(* IEC 61131-3 sources: eCockpitGit/test_project/src/%F%00 Library/%F%JSON/%POU%FB_JSONReader/%F%Structure, 12 files *)

(* ---- %METH%compareKeyName.st ---- *)
//Returns true if the inputted string is the same as the read string
METHOD compareKeyName : EStructType
VAR_INPUT
	name				:POINTER TO EASCII;
END_VAR
VAR
	posBuffer			:POINTER TO EASCII := lastKeyStart + 1;		//Buffer for key position
END_VAR
(*%!%__DELIMITER__%!%*)
IF ready AND_THEN selectedType = EStructType.object THEN
	WHILE posBuffer <= bufferADRMax DO
		CASE posBuffer^ OF
			EASCII.Null:
				IF name^ = EASCII.Null THEN
					compareKeyName		:=		lastValueType;
				END_IF
				EXIT;
			EASCII.DoubleQoute:
				IF checkNoBackSlash(checkPos:=posBuffer) THEN
					IF name^ = EASCII.Null THEN
						compareKeyName		:=		lastValueType;
					END_IF
					EXIT;
				END_IF
		END_CASE
		IF name^ <> posBuffer^ THEN
			IF posBuffer^ = EASCII.BackSlash THEN
				posBuffer				:=		posBuffer + 1;
				IF name^ <> posBuffer^ THEN
					EXIT;
				END_IF
			ELSE
				EXIT;
			END_IF
		END_IF
		name								:=		name + 1;
		posBuffer						:=		posBuffer + 1;
	END_WHILE
END_IF

(* ---- %METH%enterObjectArray.st ---- *)
//This method enters the last found object and sets it as the current object for searching
//Returns false, if not successfull
// |**Version**|**Author**| **Date** |**Changes**
// | 1         | NSN      | 04-06-18 | Creation
METHOD enterObjectArray :BOOL

(*%!%__DELIMITER__%!%*)
IF ready AND treeLevel < levelsMax THEN
	CASE lastValueType OF
		EStructType.object,EStructType.tArray:
			treeLevel			:=		treeLevel + 1;
			treeSelectedTypes[treeLevel]	:=		lastValueType;
			treeSelected[treeLevel]			:=		lastValueStart;
			treeSelectedArrayProg[treeLevel]:=		0;
			lastValueStart		:=		0;
			lastValueType		:=		EStructType.none;
			lastKeyStart		:=		0;
			enterObjectArray	:=		TRUE;
	END_CASE
END_IF

(* ---- %METH%exitObjectArray.st ---- *)
//This method exits the current object or array
//Returns none, when there are no more keys
// |**Version**|**Author**| **Date** |**Changes**
// | 1         | NSN      | 04-06-18 | Creation
METHOD exitObjectArray : BOOL
VAR
	inString		:BOOL;
	posBuffer		:POINTER TO EASCII := treeSelected[treeLevel] - 1;
	level			:WORD := 1;		//This value makes sure it doesn't return a key from inside another object
	keyFound		:BOOL;
END_VAR
(*%!%__DELIMITER__%!%*)
IF ready AND treeLevel > 1 THEN
	WHILE posBuffer >= bufferADROrg DO
		CASE posBuffer^ OF
			EASCII.DoubleQoute:
				IF checkNoBackSlash(checkPos:=posBuffer) THEN
					inString					:=		NOT(inString);
					IF keyFound AND NOT(inString) THEN
						lastKeyStart			:=		posBuffer;
					END_IF
				END_IF
			EASCII.Colon:
				IF NOT(inString) THEN
					keyFound					:=		TRUE;
				END_IF
			EASCII.CloseBraces,EASCII.SqBracketC:
				IF NOT(inString) THEN
					level						:=		level + 1;
				END_IF
			EASCII.OpenBraces,EASCII.SqBracketO,EASCII.Comma:
				IF NOT(inString) THEN
					IF level = 1 THEN
						lastValueStart			:=		treeSelected[treeLevel];
						lastValueType			:=		treeSelectedTypes[treeLevel];
						treeLevel				:=		treeLevel - 1;
						exitObjectArray			:=		TRUE;
						RETURN;
					ELSE
						level					:=		level - 1;
					END_IF
				END_IF
		END_CASE
		posBuffer								:=		posBuffer - 1;
	END_WHILE
END_IF

(* ---- %METH%exportSelection.st ---- *)
//This method outputs the start address and size of the currently selected object
//True when ok
// |**Version**|**Author**| **Date** |**Changes**
// | 1         | NSN      | 04-06-18 | Creation
METHOD exportSelection : BOOL
VAR_OUTPUT
	position		:POINTER TO EASCII;
	size			:DWORD;
END_VAR
VAR
	inString		:BOOL;
	posBuffer		:POINTER TO EASCII := treeSelected[treeLevel];
	level			:WORD;		//This value makes sure it doesn't return a key from inside another object
END_VAR
(*%!%__DELIMITER__%!%*)
IF ready AND treeLevel > 0 THEN
	position			:=		treeSelected[treeLevel];
	WHILE posBuffer < bufferADRMax DO
		CASE posBuffer^ OF
			EASCII.Null:EXIT;
			EASCII.DoubleQoute: IF checkNoBackSlash(checkPos:=posBuffer) THEN inString := NOT(inString); END_IF
			EASCII.CloseBraces,EASCII.SqBracketC: IF NOT(inString) THEN IF level > 1 THEN level := level - 1;ELSE EXIT; END_IF END_IF
			EASCII.OpenBraces,EASCII.SqBracketO: IF NOT(inString) THEN level := level + 1; END_IF
		END_CASE
		posBuffer												:=		posBuffer + 1;
	END_WHILE
	size				:=		posBuffer - position + 1;
	exportSelection		:=		TRUE;
END_IF

(* ---- %METH%findKey.st ---- *)
//This method finds the key of the given name in the object
//Returns cursor to where it was before if no tag is found
// |**Version**|**Author**| **Date** |**Changes**
// | 1         | NSN      | 04-06-18 | Creation
METHOD findKey : EStructType
VAR_INPUT
	name			:POINTER TO EASCII;		//Address of the name to find, only input string address or zero terminated byte array
END_VAR
VAR
	inString		:BOOL;
	nameBuffer		:POINTER TO EASCII;		//Buffer for cursor position
	posBuffer		:POINTER TO EASCII := treeSelected[treeLevel];
	level			:WORD;		//This value makes sure it doesn't return a key from inside another object
	foundKeyBuffer	:POINTER TO EASCII;
	slashDepth		:WORD;
END_VAR
(*%!%__DELIMITER__%!%*)
IF ready AND treeLevel > 0 AND treeSelectedTypes[treeLevel] = EStructType.object THEN
	WHILE posBuffer <= bufferADRMax DO
		CASE posBuffer^ OF
			EASCII.Null:EXIT;
			EASCII.DoubleQoute: IF checkNoBackSlash(checkPos:=posBuffer) THEN inString := NOT(inString); END_IF
			EASCII.CloseBraces,EASCII.SqBracketC: IF NOT(inString) THEN IF level > 1 THEN level := level - 1;ELSE EXIT; END_IF END_IF
			EASCII.SqBracketO: IF NOT(inString) THEN level := level + 1;END_IF
			EASCII.Comma,EASCII.OpenBraces:
				IF NOT(inString) THEN
					IF posBuffer^ = EASCII.OpenBraces THEN
						level									:=		level + 1;
					END_IF
					IF level = 1 THEN
						WHILE posBuffer <= bufferADRMax DO
							posBuffer							:=		posBuffer + 1;
							CASE posBuffer^ OF
								EASCII.Null:EXIT;
								EASCII.DoubleQoute:
									inString										:=		TRUE;
									nameBuffer										:=		name;
									foundKeyBuffer									:=		posBuffer;
									posBuffer										:=		posBuffer + 1;
									WHILE posBuffer <= bufferADRMax DO
										IF nameBuffer^ = EASCII.Null AND_THEN posBuffer^ = EASCII.DoubleQoute THEN
											WHILE posBuffer <= bufferADRMax DO
												CASE posBuffer^ OF
													EASCII.Null:EXIT;
													EASCII.DoubleQoute:
														IF checkNoBackSlash(checkPos:=posBuffer) THEN
															inString := NOT(inString);
														END_IF
													EASCII.Colon:
														IF NOT(inString) THEN
															findKey					:=		getType(valueFirstByte:=posBuffer + 1,valuePos=>lastValueStart);
															lastKeyStart			:=		foundKeyBuffer;
															lastValueType			:=		findKey;
															RETURN;
														END_IF
												END_CASE
												posBuffer							:=		posBuffer + 1;
											END_WHILE
										END_IF
										//Check for escape character
										IF nameBuffer^ = EASCII.DoubleQoute OR posBuffer^ = EASCII.BackSlash THEN
											posBuffer								:=		posBuffer + 1;
											IF posBuffer^ <> EASCII.DoubleQoute THEN
												posBuffer							:=		posBuffer - 1;
											END_IF
										END_IF
										IF posBuffer^ <> nameBuffer^ OR posBuffer^ = EASCII.Null THEN
											IF posBuffer^ = EASCII.DoubleQoute THEN
												IF checkNoBackSlash(checkPos:=posBuffer) THEN
													inString := NOT(inString);
												END_IF
											END_IF
											EXIT;
										END_IF
										nameBuffer									:=		nameBuffer + 1;
										posBuffer									:=		posBuffer + 1;
									END_WHILE
									EXIT;
							END_CASE
						END_WHILE
					END_IF
				END_IF
		END_CASE
		posBuffer																	:=		posBuffer + 1;
	END_WHILE
	findKey																			:=		EStructType.none;
END_IF

(* ---- %METH%nextArray.st ---- *)
//This method finds the next value in an array
//Returns none, when there are no more entries
// |**Version**|**Author**| **Date** |**Changes**
// | 1         | NSN      | 04-06-18 | Creation
METHOD nextArray : EStructType
VAR
	inString		:BOOL;
	posBuffer		:POINTER TO EASCII := lastValueStart;
	level			:WORD;		//This value makes sure it doesn't return a key from inside another object
END_VAR
(*%!%__DELIMITER__%!%*)
IF ready AND treeLevel > 0 AND treeSelectedTypes[treeLevel] = EStructType.tArray THEN
	IF lastValueStart = 0 THEN
		posBuffer									:=		treeSelected[treeLevel];
	ELSE
		level										:=		1;
	END_IF
	WHILE posBuffer <= bufferADRMax DO
		CASE posBuffer^ OF
			EASCII.Null:EXIT;
			EASCII.DoubleQoute: IF checkNoBackSlash(checkPos:=posBuffer) THEN inString := NOT(inString); END_IF
			EASCII.CloseBraces,EASCII.SqBracketC: IF NOT(inString) THEN IF level > 1 THEN level := level - 1;ELSE EXIT; END_IF END_IF
			EASCII.OpenBraces: IF NOT(inString) THEN level := level + 1;END_IF
			EASCII.Comma,EASCII.SqBracketO:
				IF NOT(inString) THEN
					IF posBuffer^ = EASCII.SqBracketO THEN
						level						:=		level + 1;
					END_IF
					IF level = 1 THEN
						nextArray					:=		getType(valueFirstByte:=posBuffer + 1,valuePos=>lastValueStart);
						lastValueType				:=		nextArray;
						treeSelectedArrayProg[treeLevel]	:=		treeSelectedArrayProg[treeLevel] + 1;
						RETURN;
					END_IF
				END_IF
		END_CASE
		posBuffer									:=		posBuffer + 1;
	END_WHILE
	nextArray										:=		EStructType.none;
END_IF

(* ---- %METH%nextKey.st ---- *)
//This method finds the next key/value pair in the current object
//Returns none, when there are no more keys
// |**Version**|**Author**| **Date** |**Changes**
// | 1         | NSN      | 04-06-18 | Creation
METHOD nextKey : EStructType
VAR
	inString		:BOOL;
	posBuffer		:POINTER TO EASCII := lastKeyStart;
	level			:WORD;		//This value makes sure it doesn't return a key from inside another object
	foundKeybuffer	:POINTER TO EASCII;
END_VAR
(*%!%__DELIMITER__%!%*)
IF ready AND treeLevel > 0 AND treeSelectedTypes[treeLevel] = EStructType.object THEN
	IF posBuffer = 0 THEN
		posBuffer												:=		treeSelected[treeLevel];
	ELSE
		level													:=		1;
	END_IF
	WHILE posBuffer < bufferADRMax DO
		CASE posBuffer^ OF
			EASCII.Null:EXIT;
			EASCII.DoubleQoute: IF checkNoBackSlash(checkPos:=posBuffer) THEN inString := NOT(inString); END_IF
			EASCII.CloseBraces,EASCII.SqBracketC: IF NOT(inString) THEN IF level > 1 THEN level := level - 1;ELSE EXIT; END_IF END_IF
			EASCII.SqBracketO: IF NOT(inString) THEN level := level + 1;END_IF
			EASCII.Comma,EASCII.OpenBraces:
				IF NOT(inString) THEN
					IF posBuffer^ = EASCII.OpenBraces THEN
						level												:=		level + 1;
					END_IF
					IF level = 1 THEN
						WHILE posBuffer <= bufferADRMax DO
							CASE posBuffer^ OF
								EASCII.Null:EXIT;
								EASCII.DoubleQoute:
									IF checkNoBackSlash(checkPos:=posBuffer) THEN
										inString := NOT(inString);
									END_IF
									IF foundKeybuffer = 0 THEN
										foundKeybuffer			:=		posBuffer;
									END_IF
								EASCII.Colon:
									IF NOT(inString) THEN
										nextKey					:=		getType(valueFirstByte:=posBuffer + 1,valuePos=>lastValueStart);
										lastValueType			:=		nextKey;
										lastKeyStart			:=		foundKeybuffer;
										lastKeySize				:=		TO_WORD(posBuffer - foundKeybuffer - 1);
										RETURN;
									END_IF
							END_CASE
							posBuffer							:=		posBuffer + 1;
						END_WHILE
					END_IF
				END_IF
		END_CASE
		posBuffer												:=		posBuffer + 1;
	END_WHILE
	nextKey														:=		EStructType.none;
END_IF

(* ---- %METH%readKeyName.st ---- *)
METHOD readKeyName : BOOL
VAR_INPUT
	name			:POINTER TO EASCII;		//Address of the name to find, only input string address or zero terminated byte array
	lenMax			:DWORD;
END_VAR
VAR_OUTPUT
	len				:WORD;
END_VAR
VAR
	posBuffer		:POINTER TO EASCII := lastKeyStart + 1;		//Buffer for key position
END_VAR
(*%!%__DELIMITER__%!%*)
IF ready AND lastValueType <> EStructType.none AND treeLevel > 0 THEN
	WHILE posBuffer <= bufferADRMax AND lenMax > 0 DO
		CASE posBuffer^ OF
			EASCII.Null:EXIT;
			EASCII.DoubleQoute:
				IF checkNoBackSlash(checkPos:=posBuffer) THEN
					EXIT;
				ELSE
					name			:=		name - 1;
				END_IF
		END_CASE
		name^						:=		posBuffer^;
		name						:=		name + 1;
		posBuffer					:=		posBuffer + 1;
		lenMax						:=		lenMax - 1;
	END_WHILE
	len								:=		TO_WORD(posBuffer - lastKeyStart - 1);
	name^							:=		EASCII.Null;
	readKeyName						:=		TRUE;
END_IF

(* ---- %METH%readKeyNameChar.st ---- *)
//This method returns the character of a given position from the key name
//Returns null if out of range
//Does not account for escape characters
//1 is the first character, 0 is also the first character
METHOD readKeyNameChar : EASCII
VAR_INPUT
	charNum			:WORD;		//Character number
END_VAR
VAR
	posBuffer		:POINTER TO EASCII;		//Buffer for key position
END_VAR
(*%!%__DELIMITER__%!%*)
IF ready AND lastValueType <> EStructType.none AND treeLevel > 0 AND charNum <= lastKeySize THEN
	IF charNum = 0 THEN
		posBuffer		:=		lastKeyStart + 1 + charNum;
	ELSE
		posBuffer		:=		lastKeyStart + charNum;
	END_IF
	readKeyNameChar		:=		posBuffer^;
END_IF

(* ---- %METH%readKeyNameLevel.st ---- *)
METHOD readKeyNameLevel : BOOL
VAR_INPUT
	name			:POINTER TO EASCII;		//Address of the name to find, only input string address or zero terminated byte array
	lenMax			:DWORD;
	level			:BYTE;					//The level to get from
END_VAR
VAR_OUTPUT
	len				:WORD;
END_VAR
VAR
	posBuffer		:POINTER TO EASCII;		//Buffer for key position
	inString		:BOOL;
	i				:WORD;
	arrString		:STRING(7);				//Buffer used for outputting array number
END_VAR
(*%!%__DELIMITER__%!%*)
IF ready AND level <= treeLevel AND treeLevel > 0 AND level > 0 THEN
	CASE treeSelectedTypes[level] OF
		EStructType.tArray:
			arrString						:=		FU_sConcat3(s1:='[',s2:=TO_STRING(treeSelectedArrayProg[level]),s3:=']');
			WHILE len <= 7 AND lenMax > 0 DO
				name^						:=		arrString[len];
				name						:=		name + 1;
				len							:=		len + 1;
				lenMax						:=		lenMax - 1;
				IF arrString[len] = EASCII.Null THEN
					EXIT;
				END_IF
			END_WHILE
			name^							:=		EASCII.Null;
		EStructType.object:
			IF level = treeLevel THEN
				readKeyName(name:=name,lenMax:=lenMax,len=>len);
			ELSE
				posBuffer						:=		treeSelected[level + 1] - 1;
				WHILE posBuffer > bufferADROrg DO
					IF inString THEN
						len						:=		len + 1;
					END_IF
					CASE posBuffer^ OF
						EASCII.Null:EXIT;
						EASCII.DoubleQoute:
							IF checkNoBackSlash(checkPos:=posBuffer) THEN
								IF inString THEN
									len			:=		len - 1;
									posBuffer	:=		posBuffer + 1;
									EXIT;
								ELSE
									inString	:=		TRUE;
								END_IF
							END_IF
					END_CASE
					posBuffer					:=		posBuffer - 1;
				END_WHILE
				FOR i := 1 TO len DO
					name^						:=		posBuffer^;
					name						:=		name + 1;
					lenMax						:=		lenMax - 1;
					posBuffer					:=		posBuffer + 1;
					IF lenMax = 0 THEN
						EXIT;
					END_IF
				END_FOR
				name^							:=		EASCII.Null;
				readKeyNameLevel				:=		TRUE;
			END_IF
	END_CASE
END_IF

(* ---- %METH%returnToObjectArrayStart.st ---- *)
//This method returns the cursor to the start of the json
// |**Version**|**Author**| **Date** |**Changes**
// | 1         | NSN      | 08-06-18 | Creation
METHOD returnToObjectArrayStart
(*%!%__DELIMITER__%!%*)
IF ready THEN
	lastValueStart		:=		0;
	lastValueType		:=		EStructType.none;
	lastKeyStart		:=		0;
END_IF

(* ---- %METH%returnToStart.st ---- *)
//This method returns the cursor to the start of the json
// |**Version**|**Author**| **Date** |**Changes**
// | 1         | NSN      | 08-06-18 | Creation
METHOD returnToStart
(*%!%__DELIMITER__%!%*)
IF ready THEN
	CASE buttomType OF
		EStructType.object,EStructType.tArray:
			treeLevel			:=		1;
			lastValueStart		:=		0;
			lastValueType		:=		EStructType.none;
			lastKeyStart		:=		0;
	END_CASE
END_IF
